// TIA Portal V16 export
// export: Created 2021-06-20T15:19:17.0312614Z, ExportSetting WithDefaults, DisplayName Totally Integrated Automation Portal, DisplayVersion V16 Update 4, DisplayName TIA Portal Version Control Interface, DisplayVersion V16 Update 2, DisplayName TIA Portal Openness, DisplayVersion V16 Update 4, DisplayName STEP 7 Professional, DisplayVersion V16 Update 4, DisplayName STEP 7 Safety, DisplayVersion V16, DisplayName WinCC Advanced, DisplayVersion V16 Update 4
FUNCTION "TestSuite" : Void   // FC6, F_FBD
{ S7_Optimized_Access := 'TRUE' }
VERSION : 0.1
// stored: AutoNumber true, IsIECCheckEnabled false, UDAEnableTagReadback false
   VAR_IN_OUT
      test_nop_var : Bool;
   END_VAR
BEGIN

REGION Network 1: Test No-Op
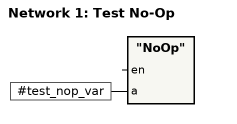
   "NoOp"("a" := #test_nop_var);
END_REGION
END_FUNCTION
